/// Saftey Lock driver.
FUNCTION_BLOCK FB_SafetyLock EXTENDS FB_ComponentBase

VAR
	/// IO structure
	stIn 				: REFERENCE TO ST_SafetyLockIn;
	stOut 				: REFERENCE TO ST_SafetyLockOut;
END_VAR

///
/// Saftey Lock driver.
/// Hannes Fuger @ asma.at		/ 09.2015
///

PROPERTY Closed : BOOL
GET
Closed := not stIn.bSaftyOK;
END_GET
END_PROPERTY

METHOD FB_init : BOOL
VAR_INPUT
	bInitRetains : BOOL; // if TRUE, the retain variables are initialized (warm start / cold start)
	bInCopyCode : BOOL;  // if TRUE, the instance afterwards gets moved into the copy code (online change)
END_VAR
eTyp := E_ComponentType.eComponentType_SafetyLock;
END_METHOD

METHOD Lock
VAR_INPUT
END_VAR
//cmd
stOut.bLock := TRUE;
END_METHOD

PROPERTY Locked : BOOL
GET
Locked := stIn.bSaftyOK AND stOut.bLock;
END_GET
END_PROPERTY

PROPERTY Opened : BOOL
GET
Opened := NOT stIn.bSaftyOK;
END_GET
END_PROPERTY

PROPERTY Referenced : BOOL
GET
Referenced:= __ISVALIDREF(stIn) AND __ISVALIDREF(stout);
END_GET
END_PROPERTY

/// Run component logic
{attribute 'object_name' := 'Run'}
METHOD Run : E_ComponentState
VAR
END_VAR
// base logic run
Run := SUPER^.Run();

stOut.bSaftyOk := stin.bSaftyOK;
END_METHOD

PROPERTY SafetyOk : BOOL
GET
SafetyOk := stIn.bSaftyOK;
END_GET
END_PROPERTY

PROPERTY SafetyOkAdr : POINTER TO BOOL
GET
SafetyOkAdr := ADR(stIn.bSaftyOK);
END_GET
END_PROPERTY

/// Set IO reference
{attribute 'object_name' := 'SetReferences'}
METHOD SetReferences
VAR_IN_OUT
	/// IO structure
	stRefIO 	: ST_SafetyLockIO;
END_VAR
stIn REF= stRefIO.stIn;
stOut REF= stRefIO.stOut;
END_METHOD

METHOD Unlock
VAR_INPUT
END_VAR
//cmd
stOut.bLock := FALSE;
END_METHOD

END_FUNCTION_BLOCK

(* stored: Version 1.1.0.1, ProductVersion 3.1.4022.12
   POU FB_SafetyLock: Id {f49f9816-ccd9-4f28-ba27-a4bc105b7a62}, SpecialFunc None
   Property Closed: Id {8e332c06-2283-43bd-add1-77c8fb609d8f}
   Get Get: Id {eca2acd8-6121-4fc1-a7b2-84b061cd3772}
   Method FB_init: Id {b92c8030-4ea8-4b89-aadb-b739f5e8b81e}
   Method Lock: Id {2b7d873a-a38e-424d-842b-af81cca30d1a}
   Property Locked: Id {edfa26f4-4d42-4d0c-9b04-3053e04f93be}
   Get Get: Id {0f61facd-a0fd-4a53-9b56-78aa4b9e7648}
   Property Opened: Id {e1bd4074-2366-485a-b902-119aa8f0012a}
   Get Get: Id {b6b91a07-b2e6-4977-9375-9ad49b32aaa2}
   Property Referenced: Id {57cd8a7d-3bc9-448b-8755-fc4ccf35c994}
   Get Get: Id {df49ae4a-98bc-4e3a-ae60-4b5fc9eae5f9}
   Method Run: Id {cf35d5e9-c2d1-45a6-b28f-a2e5485c2d67}
   Property SafetyOk: Id {a0cf24ce-6cb9-4e1c-ad34-8a37688db0d7}
   Get Get: Id {5a03da50-9366-4c01-a844-5e47b5c0cc9c}
   Property SafetyOkAdr: Id {d188a05c-38b2-4ca6-84ed-8ad6ae744b00}
   Get Get: Id {301ad23f-e96f-46c5-8a37-b0903b3cef53}
   Method SetReferences: Id {a63495bf-664d-427a-8f43-a463bf4b87c9}
   Method Unlock: Id {f280ed83-d7c7-4037-9336-4e82f5a760e4} *)
